FUNCTION CheckDivReal : REAL
VAR_INPUT
	divisor:REAL;
END_VAR

{noflow}
IF divisor = 0 THEN
	oaksGVL.udiCheckDivReal := oaksGVL.udiCheckDivReal + 1;
	CheckDivReal := 1;
ELSE
	CheckDivReal:=divisor;
END_IF;
{flow}

END_FUNCTION

(* stored: Version 1.1.0.1, ProductVersion 3.1.4022.18
   POU CheckDivReal: Id {5211caa9-16cb-4e5e-b941-1f9ffcbba7a4}, SpecialFunc CheckDivReal32 *)
